PROGRAM PRG_LivingRoom
VAR_INPUT
END_VAR
VAR_OUTPUT
END_VAR
VAR
	fbLivingRoom					: FB_LivingRoom;
END_VAR

(*
****************************************************************************************************************************

****************************************************************************************************************************

Erstellt:       FÖB      20.09.2022
 
Geändert:       

****************************************************************************************************************************
Was man wissen sollte:

****************************************************************************************************************************
*)

//**************************************************************************************************************************
// Aufruf Ablaufsteuerung
//**************************************************************************************************************************

fbLivingRoom(
	ixErrorAcknowledge:= , 
	ixAcknowledgePulse:= , 
	sHmi:= GVL_HMI.sRooms.sLivingRoom, 
	sMqttClient:= GVL_Mqtt.sClient, 
	sStatusDevices:= GVL_Devices.sStatus);

END_PROGRAM

(* stored: Version 1.1.0.1, ProductVersion 3.1.4024.12
   POU PRG_LivingRoom: Id {bd6078c0-a02d-48fd-bce0-efedf8a47448}, SpecialFunc None *)
